Fanuc KAREL source: KA00217.KL

PROGRAM KA00217
%NOLOCKGROUP
VAR
  SRC: ARRAY[4] OF JOINTPOS
  DST: ARRAY[4] OF INTEGER
BEGIN
  DST = SRC
END KA00217
